(* PLC project OOP_Curso, Beckhoff Automation GmbH TwinCAT PLC Control 3.5.13.21 *)
(* stored: creationDateTime 2023-06-23T16:27:20.9848655, modificationDateTime 2023-06-23T16:27:20.9848655 *)

PROGRAM _19_ExST
VAR
	myVar: INT;
	myVar1: INT;
	myVar2: INT;
	
	b: BOOL;
	i: INT;	
	btrig : F_TRIG;
	counter: INT;
	
	bVar1: BOOL;
	bVar2: BOOL;
	
	bVar11: BOOL;
	bVar22: BOOL;
	
	bVar: BOOL;
	bVarS: BOOL;
	bVarR: BOOL;
	
	bVara: BOOL;
	bVarb: BOOL;
	bVarc: BOOL;
	
	bMyVar1: BOOL;
	bMyVar2: BOOL;
	bmyTimer : BOOL;
	myTimer : TON;
	

END_VAR

            myVar := myVar1 := myVar2 + 26 ; 

IF b := (i = 1) THEN i := i + 1; END_IF	

btrig(CLK:=b);

IF btrig.Q THEN
	counter := counter + 1;
END_IF

bVar1 S= bVar2;

bVar11 R= bVar22;

bVar S= bVarS R= bVarR;

bVara R= bVarb S= bVarc;

myTimer(IN:= bmyTimer , PT:= T#2S );

bMyVar1 S= bMyVar2 R= myTimer.Q;
          
END_PROGRAM
